// TIA Portal V19 export
TYPE "LAF_typeDevDiagInternal"
TITLE = Structure device diag internal / Struktur device diag intern
// This data type contains internal data of the function block which is not used for display on the HMI.  
// 
// **PLC Data types**  
// * [LAF_typeDevDiagNoOfDevices](../Library%20Types/LAF_typeDevDiagNoOfDevices.htm)  
// * [LAF_typeDevDiagHwAddress](../Library%20Types/LAF_typeDevDiagHwAddress.htm)
// Profinet device Diagnose
// stored: Access Published
   STRUCT
      localProfinetSystem { ExternalAccessible := 'False'; ExternalVisible := 'False'; ExternalWritable := 'False'} : HW_IOSYSTEM;   // Profinet System / Profinet system
      maxDevices { ExternalAccessible := 'False'; ExternalVisible := 'False'; ExternalWritable := 'False'} : DInt;   // Max. number of devices to be evaluated / Max. Anzahl Devices zum auswerten
      maxModules { ExternalAccessible := 'False'; ExternalVisible := 'False'; ExternalWritable := 'False'} : DInt;   // Max. number of modules to be evaluated / Max. Anzahl Module zum auswerten
      numberDevices { ExternalAccessible := 'False'; ExternalVisible := 'False'; ExternalWritable := 'False'} : "LAF_typeDevDiagNoOfDevices";   // Via "DevicesStates" ausgewertete Informationen / Via "DevicesStates" evaluated info
      hwAddress { ExternalAccessible := 'False'; ExternalVisible := 'False'; ExternalWritable := 'False'} : Array[0..256] of "LAF_typeDevDiagHwAddress";   // Device HWTYPE
   END_STRUCT;
END_TYPE
